Fanuc KAREL source: kc00051.KL

-- PROVISIONAL review KL for V1013-1; original PC SHA256 bb74615bb33ed69a66ebe32ea31f311a1e5fbbaf79cd167ad508f4c34767e3f7
-- Incomplete behavior may be omitted. Consult companion uncertainty JSON. Do not deploy.
PROGRAM KC00051
%NOLOCKGROUP
BEGIN
  -- UNRESOLVED_PC offsets 5-29; opcodes 27,22,22,2A,22,31
  -- UNRESOLVED_PC offsets 34-38; opcodes 7F
END KC00051
